(* IEC 61131-3 sources: ELE/滚筒阻挡工程/SBR程序块, 6 files *)

(* ---- SBR_01_通用FB库.st ---- *)
(* ════════════════════════════════════════════════════════════════════
   SBR_01 通用 FB 库
   FB 接口/内部变量对应 变量表\FbTable_*.csv (类别 IN/OUT/INOUT/VAR)
   ════════════════════════════════════════════════════════════════════ *)

(* ── FB1 故障锁存: 边沿置位, 故障源消除+复位命令才清除 (细则2) ── *)
FUNCTION_BLOCK FB_AlarmLatch
VAR_INPUT
    FaultSrc : BOOL;        (* 故障源输入(电平) *)
    ResetCmd : BOOL;        (* 复位命令(外部已做上升沿) *)
END_VAR
VAR_OUTPUT
    AlarmOut : BOOL;        (* 报警锁存输出 *)
END_VAR
VAR
    bLatched : BOOL;        (* 内部锁存位 *)
END_VAR
IF FaultSrc THEN
    bLatched := TRUE;
ELSIF ResetCmd AND (NOT FaultSrc) THEN
    bLatched := FALSE;      (* 复位需故障源已消除, 不允许带故障复位 *)
END_IF;
AlarmOut := bLatched;

(* ── FB2 电辊筒: 方向互锁 + 三档速度经输入传入 (禁止 FB 内全局常量) ── *)
FUNCTION_BLOCK FB_Roller
VAR_INPUT
    FwdInput  : BOOL;       (* 正转启动 *)
    RevInput  : BOOL;       (* 反转启动(与正转互锁) *)
    SpeedLevel : INT;       (* 速度档(1低/2中/3高) *)
    SpeedLow  : INT;        (* 低速档百分比 *)
    SpeedMid  : INT;        (* 中速档百分比 *)
    SpeedHigh : INT;        (* 高速档百分比 *)
    Enable    : BOOL;       (* 运行许可(RunOK 门控) *)
    Reset     : BOOL;       (* 故障复位 *)
END_VAR
VAR_OUTPUT
    FwdOut    : BOOL;       (* 正转输出 *)
    RevOut    : BOOL;       (* 反转输出(预留) *)
    Error     : BOOL;       (* 故障标志 *)
END_VAR
VAR
    bRun   : BOOL;          (* 内部运行状态 *)
    iSpeed : INT;           (* 内部当前速度 *)
END_VAR
(* 复位清故障 *)
IF Reset THEN
    Error := FALSE;
END_IF;
(* 无许可强制停 (显式切断 细则13) *)
IF NOT Enable THEN
    bRun := FALSE;
END_IF;
(* 方向命令: 同发视为无效防误动, 单向有效 (互锁细则7) *)
IF FwdInput AND (NOT RevInput) THEN
    bRun := TRUE;
ELSIF RevInput AND (NOT FwdInput) THEN
    bRun := TRUE;
ELSIF (NOT FwdInput) AND (NOT RevInput) THEN
    bRun := FALSE;
END_IF;
(* 速度档查表 *)
CASE SpeedLevel OF
    1: iSpeed := SpeedLow;
    2: iSpeed := SpeedMid;
    3: iSpeed := SpeedHigh;
ELSE
    iSpeed := 0;
END_CASE;
(* 输出: 许可门控 + 反向互斥 *)
FwdOut := bRun AND Enable AND (NOT RevInput) AND (iSpeed > 0);
RevOut := FALSE;

(* ---- SBR_04_模式管理.st ---- *)
(* ════════════════════════════════════════════════════════════════════
   SBR_04 模式管理
   手自动旋钮电平采集 + 切换瞬间清零 (互斥 细则7, 边沿时序 细则6)
   ════════════════════════════════════════════════════════════════════ *)

(* 先比较后更新: 检测到模式切换 -> 清自动步/手动翻转/命令量, 防残留误动作 *)
IF bModeAuto <> in_ModeAuto THEN
    con_AutoStep      := 0;
    bManBlockTgl      := FALSE;
    con_BlockUpCmd    := FALSE;
    con_RollerRunCmd  := FALSE;
END_IF;

(* 模式电平: TRUE=自动 FALSE=手动 *)
bModeAuto := in_ModeAuto;

(* ---- SBR_05_手动控制.st ---- *)
(* ════════════════════════════════════════════════════════════════════
   SBR_05 手动控制
   手动模式: 本地复位键翻转阻挡 + 上位机远程命令(通讯字表 写区)
   优先级: 远程命令 > 本地按键; 通讯丢失时远程命令失效 (细则9)
   与 SBR_06 自动控制按 bModeAuto 互斥, 每周期只有一方写命令量 (细则7)
   ════════════════════════════════════════════════════════════════════ *)
IF (NOT bModeAuto) AND bRunOK THEN
    (* ── 滚筒: 远程正转/停止 (写1触发, 停止优先; 无远程命令时保持停) ── *)
    IF con_CommLost THEN
        con_RollerRunCmd := FALSE;
    ELSIF host_Send_RollerStop = 1 THEN
        con_RollerRunCmd := FALSE;
    ELSIF host_Send_RollerFwd = 1 THEN
        con_RollerRunCmd := TRUE;
    ELSE
        con_RollerRunCmd := FALSE;
    END_IF;

    (* ── 阻挡: 远程升/降优先, 无远程命令时本地复位键翻转仍可用 ── *)
    IF con_CommLost THEN
        con_BlockUpCmd := FALSE;
    ELSIF host_Send_BlockUp = 1 THEN
        con_BlockUpCmd := TRUE;
    ELSIF host_Send_BlockDn = 1 THEN
        con_BlockUpCmd := FALSE;
    ELSE
        r_ManBlock(CLK := in_Reset);
        IF r_ManBlock.Q THEN
            bManBlockTgl := NOT bManBlockTgl;
        END_IF;
        con_BlockUpCmd := bManBlockTgl;
    END_IF;
ELSE
    bManBlockTgl := FALSE;
END_IF;

(* ---- SBR_06_自动控制.st ---- *)
(* ════════════════════════════════════════════════════════════════════
   SBR_06 自动控制 (步进状态机)
   步0 待机启动 -> 步1 阻挡输送(定时+磁开确认) -> 步2 放行(定时+磁开确认) -> 回步1
   气缸到位看门狗: 超时未到位 -> con_CylTimeout 接报警锁存闭环
   与 SBR_05 按 bModeAuto 互斥; 非自动/许可丢失时显式切断全部命令 (细则13)
   ════════════════════════════════════════════════════════════════════ *)
IF bModeAuto AND bRunOK THEN
    CASE con_AutoStep OF
        0:  (* 待机: 滚筒先转, 进入输送节拍 *)
            con_BlockUpCmd   := FALSE;
            con_RollerRunCmd := TRUE;
            con_AutoStep     := 1;

        1:  (* 阻挡输送: 升阻挡截停工件, 滚筒持续 *)
            con_BlockUpCmd   := TRUE;
            con_RollerRunCmd := TRUE;
            ton_BlockHold(IN := TRUE, PT := BLOCK_HOLD_TIME);
            ton_CylWatch(IN  := TRUE, PT := CYL_TIMEOUT);
            IF ton_CylWatch.Q AND (NOT in_BlockUpSns) THEN
                con_CylTimeout := TRUE;      (* 升不到位 -> 报警源, 锁存于安全回路 *)
            END_IF;
            IF in_BlockUpSns AND ton_BlockHold.Q THEN
                con_AutoStep := 2;           (* 磁开确认 + 保持时间到 -> 放行 *)
                ton_BlockHold(IN := FALSE, PT := BLOCK_HOLD_TIME);
                ton_CylWatch(IN  := FALSE, PT := CYL_TIMEOUT);
            END_IF;

        2:  (* 放行: 降阻挡放行工件, 滚筒持续 *)
            con_BlockUpCmd   := FALSE;
            con_RollerRunCmd := TRUE;
            ton_PassTime(IN  := TRUE, PT := BLOCK_PASS_TIME);
            ton_CylWatch(IN  := TRUE, PT := CYL_TIMEOUT);
            IF ton_CylWatch.Q AND (NOT in_BlockDnSns) THEN
                con_CylTimeout := TRUE;      (* 降不到位 -> 报警源 *)
            END_IF;
            IF in_BlockDnSns AND ton_PassTime.Q THEN
                con_AutoStep := 1;           (* 磁开确认 + 放行时间到 -> 下一节拍 *)
                con_CycleCnt := con_CycleCnt + 1;   (* 完成一次放行: 节拍计数+1(掉电保持) *)
                ton_PassTime(IN := FALSE, PT := BLOCK_PASS_TIME);
                ton_CylWatch(IN  := FALSE, PT := CYL_TIMEOUT);
            END_IF;

        ELSE
            con_AutoStep := 0;               (* 非法步号兜底回待机 *)
    END_CASE;
ELSE
    (* 显式安全切断: 手动模式/急停/报警/许可丢失 -> 全部命令清零+计时器复位 (细则13) *)
    con_AutoStep     := 0;
    con_BlockUpCmd   := FALSE;
    con_RollerRunCmd := FALSE;
    con_CylTimeout   := FALSE;
    ton_BlockHold(IN := FALSE, PT := BLOCK_HOLD_TIME);
    ton_PassTime(IN  := FALSE, PT := BLOCK_PASS_TIME);
    ton_CylWatch(IN  := FALSE, PT := CYL_TIMEOUT);
END_IF;

(* ---- SBR_07_输出刷新.st ---- *)
(* ════════════════════════════════════════════════════════════════════
   SBR_07 输出刷新 (主调度最后一步)
   辊筒 FB 调用 + 物理输出统一刷新: 先显式默认, 再经 RunOK 许可门控 (细则13/14)
   ════════════════════════════════════════════════════════════════════ *)

(* 滚筒 FB: 本工程单速正向, 三档速度经输入参数传入 (速度档不作 FB 内常量) *)
Roller_1(FwdInput   := con_RollerRunCmd,
         RevInput   := FALSE,
         SpeedLevel := 1,
         SpeedLow   := 100,
         SpeedMid   := 75,
         SpeedHigh  := 50,
         Enable     := bRunOK,
         Reset      := con_ResetCmd);

(* 物理输出刷新: 显式默认 FALSE, 无许可强制安全态 *)
out_RollerRun := FALSE;
out_BlockUp   := FALSE;
IF bRunOK THEN
    out_RollerRun := Roller_1.FwdOut;
    out_BlockUp   := con_BlockUpCmd;
END_IF;

(* ---- SBR_host_上位机通讯.st ---- *)
(* ════════════════════════════════════════════════════════════════════
   SBR_host 上位机通讯 (Modbus TCP, 字表见 通讯字表.csv)
   状态映射回写 + 命令清0回执 + 双心跳看门狗 (心跳入/出向分离 细则9)
   ════════════════════════════════════════════════════════════════════ *)

(* ── 入向心跳: 变化检测 -> 看门狗; 超时判通讯丢失 (接 RunOK 联锁) ── *)
IF host_Send_Heart <> con_HeartPrev THEN
    con_HeartPrev := host_Send_Heart;        (* 检测到变化: 复位看门狗输入 *)
END_IF;
ton_CommWatch(IN := NOT (host_Send_Heart <> con_HeartPrev), PT := COMM_HEART_TIMEOUT);
IF ton_CommWatch.Q THEN
    con_CommLost := TRUE;                    (* 超时未变化 -> 通讯丢失 *)
ELSE
    con_CommLost := FALSE;
END_IF;

(* ── 出向心跳: 每 COMM_HEART_TICK 自增1 写回上位机 (PLC存活示警) ── *)
ton_HeartTick(IN := TRUE, PT := COMM_HEART_TICK);
IF ton_HeartTick.Q THEN
    con_HeartOut := con_HeartOut + 1;
END_IF;

(* ── 命令清0回执协议: 动作确认后由 PLC 清零命令字, 防重复触发 ──
   阻挡升降: 到位(磁开)即清 | 报警复位: 边沿消费后清 | 滚筒停止: 停稳后清 *)
IF in_BlockUpSns AND (host_Send_BlockUp = 1) THEN
    host_Send_BlockUp := 0;
END_IF;
IF in_BlockDnSns AND (host_Send_BlockDn = 1) THEN
    host_Send_BlockDn := 0;
END_IF;
IF r_HostReset.Q THEN
    host_Send_AlarmReset := 0;
END_IF;
IF (host_Send_RollerStop = 1) AND (NOT Roller_1.FwdOut) THEN
    host_Send_RollerStop := 0;
END_IF;

(* ── 状态区回写 (INT 化, BOOL->0/1 显式转换) ── *)
host_Rcv_Mode     := SEL(bModeAuto, 0, 1);
host_Rcv_Estop    := SEL(bEstopPressed, 0, 1);
host_Rcv_Alarm    := SEL(con_Alarm, 0, 1);
host_Rcv_Running  := SEL(Roller_1.FwdOut, 0, 1);
host_Rcv_BlockUp  := SEL(in_BlockUpSns, 0, 1);
host_Rcv_AutoStep := con_AutoStep;
host_Rcv_CycleCnt := con_CycleCnt;
host_Rcv_HeartOut := con_HeartOut;
